RoboDK station: New Station.rdk

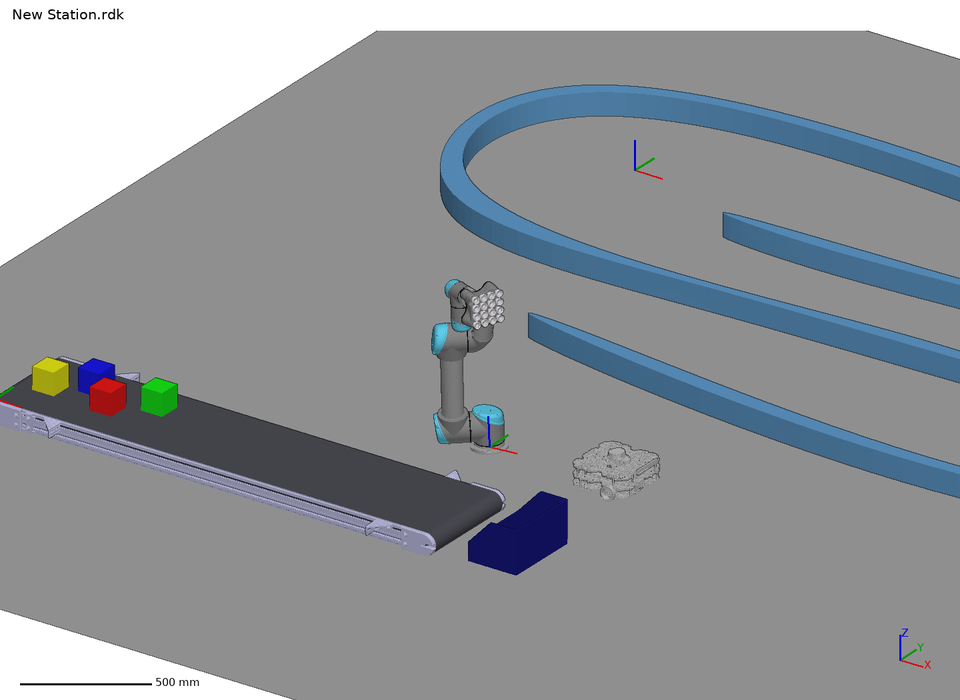
[picture v0: the station drawn from its stored meshes, robots at their saved joint values, targets as dots, program paths as lines]
Station New Station (saved by RoboDK 5.7.4). Poses are relative to the parent item; angles as X-Y-Z fixed-axis rotations.
  - frame MainFrame at (0, 0, 0) mm
  - frame UR5 Base at (920, -2280, 0) mm, rotated rx 0 ry -2.58 rz 0 deg
    - robot UR5: 6 axes
        modified DH rows (alpha deg, a mm, theta deg, d mm): 0, 0, 0, 89.2; 90, 0, 180, 0; 0, 425, 0, 0; 0, 392, 0, 109.3; -90, 0, 0, 94.75; 90, 0, 180, 82.5
        joint limits [-360, -360, -360, -360, -360, -360] to [360, 360, 360, 360, 360, 360]; home [0, -90, -90, 0, 90, 0]; saved at [-51.097, -102.135, -40.746, -37.106, 119.007, 0.649]
      - tool OnRobot VG10 Vacuum Gripper, TCP at (0, 0, 130.9) mm, size 145.4 x 145.4 x 118.3 mm
  - object Floor at (0, -3000, 0) mm, size 3000 x 3000 x 0 mm, geometry from Floor (1).sld
  - object Floor at (3000, -3000, 0) mm, size 3000 x 3000 x 0 mm, geometry from Floor (1).sld
  - object Floor at (0, 0, 0) mm, size 3000 x 3000 x 0 mm, geometry from Floor (1).sld
  - object Floor at (3000, 0, 0) mm, size 3000 x 3000 x 0 mm, geometry from Floor (1).sld
  - object Bin Red at (2930, 150, 0) mm, rotated rx 0 ry 0 rz -180 deg, size 225 x 337.5 x 191.2 mm, geometry from Bin-Red.sld
  - object Bin Blue at (1420, -2800, 0) mm, rotated rx 0 ry 0 rz -180 deg, size 225 x 337.5 x 191.2 mm, geometry from Bin-Blue.sld
  - object turtlebot3_waffle (1) at (1500, -2270, 20) mm, size 280.7 x 305.1 x 138.1 mm, geometry from turtlebot3_waffle (1).step
  - frame Conveyor Belt (2m) Base at (-740, -3190, 100) mm
    - robot Conveyor Belt (2m): 1 axes
        modified DH rows (alpha deg, a mm, theta deg, d mm): 0, 0, 0, 0 linear
        base shift (0, 0, 0) mm, rotated rx 0 ry 90 rz 0 deg
        joint limits [-500000] to [500000]; home [0]; saved at [0]
    - object Red at (400, 180, 0) mm, size 100 x 100 x 100 mm, geometry from Red.step
    - object Yellow at (120, 200, 0) mm, size 100 x 100 x 100 mm, geometry from Yellow.step
    - object Green at (560, 290, 0) mm, size 100 x 100 x 100 mm, geometry from Green.step
    - object Blue at (270, 290, 0) mm, size 100 x 100 x 100 mm, geometry from Blue.step
    - object path at (6000, 2000, 0) mm, size 3159.6 x 1446.5 x 100 mm, geometry from path.step
    - object path2 at (-1250, 2930, 40) mm, rotated rx 0 ry 0 rz 180 deg, size 3159.6 x 1446.5 x 100 mm, geometry from path.step
